INTERFACE I_Command EXTENDS I_Disposable

METHOD Execute
VAR_INPUT
END_VAR
END_METHOD

END_INTERFACE

(* stored: Version 1.1.0.1, ProductVersion 3.1.4024.12
   Itf I_Command: Id {5482795c-4fc0-4be1-b623-899f29e63002}
   Method Execute: Id {cd320ce1-cc3a-4e76-811c-b70da7184772} *)
